// TwinCAT 3 PLC project TrafficLightLibPLC
// Title: TrafficControlLib
// Company: TrafficLightProject AG
// ProjectVersion: 0.5.0
// ProgramVersion: 3.1.4024.0
// libraries:
//   Tc2_Standard, * (Beckhoff Automation GmbH)
//   Tc2_System, * (Beckhoff Automation GmbH)
//   Tc3_Module, * (Beckhoff Automation GmbH)
//   TcUnit,1.3.1,www.tcunit.org
// project tree:
//   DUTs/ E_LightState.TcDUT, E_Phase.TcDUT
//   Interfaces/ ITrafficLight.TcIO
//   / PlcTask.TcTTO
//   POUs/ FB_Intersection.TcPOU, FB_TrafficLight.TcPOU
//   Test/ FB_Intersection_Test.TcPOU, FB_MockLight.TcPOU, FB_TrafficLight_Test.TcPOU, PRG_TEST.TcPOU
// (motion and I/O tree: see PLC project trafficlightappplc)
// real-time tasks:
//   TASK PlcTask: cycle T#10ms, priority 20, ADS port 350
//   TASK PlcTask1: cycle T#10ms, priority 21, ADS port 351

CONFIGURATION TrafficLightLibPLC
    RESOURCE PLC ON TwinCAT3
        TASK PlcTask(INTERVAL := T#10ms, PRIORITY := 21);
        PROGRAM PRG_TEST WITH PlcTask : PRG_TEST;
    END_RESOURCE
END_CONFIGURATION

// ---- DUTs/E_LightState.TcDUT
{attribute 'qualified_only'}
{attribute 'strict'}
TYPE E_LightState :
(
    Red,
    RedAmber,
    Green,
    Amber
) := Red;
END_TYPE

// ---- DUTs/E_Phase.TcDUT
{attribute 'qualified_only'}
{attribute 'strict'}
TYPE E_Phase :
(
    AllRed,                 // startup and clearance — the safe state
    NorthSouthFlowing,
    NorthSouthClearing,
    EastWestFlowing,
    EastWestClearing
) := AllRed;
END_TYPE

// ---- Interfaces/ITrafficLight.TcIO
INTERFACE ITrafficLight

PROPERTY CurrentState  : E_LightState
GET
END_GET
SET
END_SET
END_PROPERTY

END_INTERFACE

// ---- Test/PRG_TEST.TcPOU
PROGRAM PRG_TEST
VAR
	fbTrafficLightTest : FB_TrafficLight_Test;
	fbIntersectionTest  : FB_Intersection_Test;
END_VAR

TcUnit.RUN();

END_PROGRAM

// ---- Test/FB_TrafficLight_Test.TcPOU
FUNCTION_BLOCK FB_TrafficLight_Test EXTENDS TcUnit.FB_TestSuite
VAR
END_VAR

NewLightStartsInRed();
LightCyclesThroughFullSequence();

METHOD PRIVATE NewLightStartsInRed
VAR
	light       : FB_TrafficLight;
    actualState : E_LightState;
END_VAR
TEST('NewLightStartsInRed');

actualState := light.CurrentState;   // read the property into a variable first

AssertEquals_INT(
    Expected := TO_INT(E_LightState.Red),
    Actual   := TO_INT(actualState),
    Message  := 'A new light should start in RED');

TEST_FINISHED();
END_METHOD

END_FUNCTION_BLOCK

// ---- POUs/FB_TrafficLight.TcPOU
FUNCTION_BLOCK FB_TrafficLight IMPLEMENTS ITrafficLight
VAR
	_state : E_LightState := E_LightState.Red;
END_VAR

{warning 'add property implementation'}
PROPERTY CurrentState : E_LightState
GET
CurrentState := _state;
END_GET
END_PROPERTY

METHOD PUBLIC SetState
VAR_INPUT
	newState : E_LightState;
END_VAR
_state := newState;
END_METHOD

END_FUNCTION_BLOCK

// ---- Test/FB_Intersection_Test.TcPOU
FUNCTION_BLOCK FB_Intersection_Test EXTENDS TcUnit.FB_TestSuite
VAR
END_VAR

NewIntersectionStartsInAllRed();
IntersectionAdvancesThroughPhasesInOrder();
NorthSouthFlowingShowsNsGreenEwRed();
NeverTwoGreensAcrossFullCycle();
ManualRequestAdvancesPhase();
UpdateReportsTrueWhenItAdvances();
UpdateReportsFalseWithoutEdge();

METHOD PRIVATE IntersectionAdvancesThroughPhasesInOrder
VAR
	nsLight      : FB_TrafficLight;
    ewLight      : FB_TrafficLight;
    intersection : FB_Intersection(nsLight := nsLight, ewLight := ewLight);
END_VAR
TEST('IntersectionAdvancesThroughPhasesInOrder');

// starts AllRed
AssertEquals_INT(
    Expected := TO_INT(E_Phase.AllRed),
    Actual   := TO_INT(intersection.CurrentPhase),
    Message  := 'Should start AllRed');

intersection.Advance();           
AssertEquals_INT(
    Expected := TO_INT(E_Phase.NorthSouthFlowing),
    Actual   := TO_INT(intersection.CurrentPhase),
    Message  := 'AllRed should advance to NorthSouthFlowing');

intersection.Advance();
AssertEquals_INT(
    Expected := TO_INT(E_Phase.NorthSouthClearing),
    Actual   := TO_INT(intersection.CurrentPhase),
    Message  := 'NorthSouthFlowing should advance to NorthSouthClearing');

intersection.Advance();
AssertEquals_INT(
    Expected := TO_INT(E_Phase.EastWestFlowing),
    Actual   := TO_INT(intersection.CurrentPhase),
    Message  := 'NorthSouthClearing should advance to EastWestFlowing');

intersection.Advance();
AssertEquals_INT(
    Expected := TO_INT(E_Phase.EastWestClearing),
    Actual   := TO_INT(intersection.CurrentPhase),
    Message  := 'EastWestFlowing should advance to EastWestClearing');

intersection.Advance();
AssertEquals_INT(
    Expected := TO_INT(E_Phase.NorthSouthFlowing),
    Actual   := TO_INT(intersection.CurrentPhase),
    Message  := 'EastWestClearing should wrap to NorthSouthFlowing (not AllRed)');

TEST_FINISHED();
END_METHOD

METHOD PRIVATE ManualRequestAdvancesPhase
VAR
	nsLight      : FB_TrafficLight;
    ewLight      : FB_TrafficLight;
    intersection : FB_Intersection(nsLight := nsLight, ewLight := ewLight);
END_VAR
TEST('ManualRequestAdvancesPhase');

// starts in AllRed; simulate a button press (rising edge)
intersection.Update(bManualStepRequest := FALSE);   // establish low baseline
intersection.Update(bManualStepRequest := TRUE);    // rising edge -> advance

AssertEquals_INT(
    Expected := TO_INT(E_Phase.NorthSouthFlowing),
    Actual   := TO_INT(intersection.CurrentPhase),
    Message  := 'A manual request should advance out of AllRed');

TEST_FINISHED();
END_METHOD

METHOD PRIVATE NeverTwoGreensAcrossFullCycle
VAR
	nsLight      : FB_TrafficLight;
    ewLight      : FB_TrafficLight;
    intersection : FB_Intersection(nsLight := nsLight, ewLight := ewLight);
    i            : INT;
    nsGreen      : BOOL;
    ewGreen      : BOOL;
END_VAR
TEST('NeverTwoGreensAcrossFullCycle');

// Walk several full cycles; the safety rule must hold at every step.
FOR i := 1 TO 12 DO
    intersection.Advance();

    nsGreen := (intersection.NorthSouthState = E_LightState.Green);
    ewGreen := (intersection.EastWestState  = E_LightState.Green);

    AssertFalse(
        Condition := (nsGreen AND ewGreen),
        Message   := 'Both directions must never be green at once');
END_FOR

TEST_FINISHED();
END_METHOD

METHOD PRIVATE NewIntersectionStartsInAllRed
VAR
	nsLight      : FB_TrafficLight;
    ewLight      : FB_TrafficLight;
    intersection : FB_Intersection(nsLight := nsLight, ewLight := ewLight);
END_VAR
TEST('NewIntersectionStartsInAllRed');

AssertEquals_INT(
    Expected := TO_INT(E_Phase.AllRed),
    Actual   := TO_INT(intersection.CurrentPhase),
    Message  := 'A new intersection should start in AllRed for safety');

TEST_FINISHED();
END_METHOD

METHOD PRIVATE NorthSouthFlowingShowsNsGreenEwRed
VAR
	nsLight      : FB_TrafficLight;
    ewLight      : FB_TrafficLight;
    intersection : FB_Intersection(nsLight := nsLight, ewLight := ewLight);
END_VAR
TEST('NorthSouthFlowingShowsNsGreenEwRed');

intersection.Advance();   // AllRed -> NorthSouthFlowing

AssertEquals_INT(
    Expected := TO_INT(E_LightState.Green),
    Actual   := TO_INT(intersection.NorthSouthState),
    Message  := 'NS should be GREEN in NorthSouthFlowing');

AssertEquals_INT(
    Expected := TO_INT(E_LightState.Red),
    Actual   := TO_INT(intersection.EastWestState),
    Message  := 'EW should be RED in NorthSouthFlowing');

TEST_FINISHED();
END_METHOD

METHOD PRIVATE UpdateReportsFalseWithoutEdge
VAR
	nsLight      : FB_TrafficLight;
    ewLight      : FB_TrafficLight;
    intersection : FB_Intersection(nsLight := nsLight, ewLight := ewLight);
    didAdvance   : BOOL;
END_VAR
TEST('UpdateReportsFalseWithoutEdge');

didAdvance := intersection.Update(bManualStepRequest := FALSE);  // no request

AssertFalse(
    Condition := didAdvance,
    Message   := 'Update should report FALSE when there is no manual request');

TEST_FINISHED();
END_METHOD

METHOD PRIVATE UpdateReportsTrueWhenItAdvances
VAR
	nsLight      : FB_TrafficLight;
    ewLight      : FB_TrafficLight;
    intersection : FB_Intersection(nsLight := nsLight, ewLight := ewLight);
    didAdvance   : BOOL;
END_VAR
TEST('UpdateReportsTrueWhenItAdvances');

intersection.Update(bManualStepRequest := FALSE);              // baseline low
didAdvance := intersection.Update(bManualStepRequest := TRUE); // rising edge

AssertTrue(
    Condition := didAdvance,
    Message   := 'Update should report TRUE on the scan it advances');

TEST_FINISHED();
END_METHOD

END_FUNCTION_BLOCK

// ---- POUs/FB_Intersection.TcPOU
FUNCTION_BLOCK FB_Intersection
VAR
    _phase : E_Phase := E_Phase.AllRed;

    // Lights are now INJECTED, not created here
    _nsLight : ITrafficLight;
    _ewLight : ITrafficLight;

    _rtrigManual : R_TRIG;
END_VAR

METHOD PUBLIC Advance
VAR
END_VAR
// Normal-mode behavior for now.
// A control-mode CASE (Emergency, NightFlash, Manual) would wrap this later.
RunNormalCycle();
ApplyPhaseToLights();
END_METHOD

METHOD PRIVATE ApplyPhaseToLights
VAR_INPUT
END_VAR
CASE _phase OF

    E_Phase.AllRed:
        _nsLight.CurrentState := E_LightState.Red;
        _ewLight.CurrentState := E_LightState.Red;

    E_Phase.NorthSouthFlowing:
        _nsLight.CurrentState := E_LightState.Green;
        _ewLight.CurrentState := E_LightState.Red;

    E_Phase.NorthSouthClearing:
        _nsLight.CurrentState := E_LightState.Amber;
        _ewLight.CurrentState := E_LightState.Red;

    E_Phase.EastWestFlowing:
        _nsLight.CurrentState := E_LightState.Red;
        _ewLight.CurrentState := E_LightState.Green;

    E_Phase.EastWestClearing:
        _nsLight.CurrentState := E_LightState.Red;
        _ewLight.CurrentState := E_LightState.Amber;

END_CASE
END_METHOD

PROPERTY CurrentPhase : E_Phase
GET
CurrentPhase := _phase;
END_GET
END_PROPERTY

PROPERTY EastWestState : E_LightState
GET
EastWestState := _ewLight.CurrentState;
END_GET
END_PROPERTY

METHOD FB_init : BOOL
VAR_INPUT
    bInitRetains : BOOL;
    bInCopyCode  : BOOL;
    nsLight      : ITrafficLight;   // injected
    ewLight      : ITrafficLight;   // injected
END_VAR
_nsLight := nsLight;
_ewLight := ewLight;
END_METHOD

PROPERTY NorthSouthState : E_LightState
GET
NorthSouthState := _nsLight.CurrentState;
END_GET
END_PROPERTY

METHOD PRIVATE RunNormalCycle
VAR
END_VAR
CASE _phase OF

    E_Phase.AllRed:
        _phase := E_Phase.NorthSouthFlowing;

    E_Phase.NorthSouthFlowing:
        _phase := E_Phase.NorthSouthClearing;

    E_Phase.NorthSouthClearing:
        _phase := E_Phase.EastWestFlowing;

    E_Phase.EastWestFlowing:
        _phase := E_Phase.EastWestClearing;

    E_Phase.EastWestClearing:
        _phase := E_Phase.NorthSouthFlowing;  

END_CASE
END_METHOD

METHOD PUBLIC Update : BOOL
VAR_INPUT
	bManualStepRequest : BOOL;
END_VAR
// A rising edge on the manual request advances the intersection once.
// Reuses Advance() so phase AND lights update through the single code path.
_rtrigManual(CLK := bManualStepRequest);

IF (_rtrigManual.Q) THEN
    Advance();
    Update := TRUE;      // report that a manual advance happened
ELSE
    Update := FALSE;
END_IF
END_METHOD

END_FUNCTION_BLOCK

// ---- Test/FB_MockLight.TcPOU
FUNCTION_BLOCK FB_MockLight IMPLEMENTS ITrafficLight
VAR
	_state : E_LightState := E_LightState.Red;
END_VAR

{warning 'add property implementation'}
PROPERTY CurrentState : E_LightState
GET
CurrentState := _state;
END_GET
SET
_state := CurrentState;
END_SET
END_PROPERTY

END_FUNCTION_BLOCK
